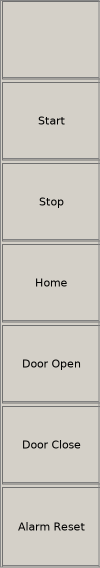
VISUALIZATION SideBar  // 100x568
    Button (2,1 99x78), colour toggle: GVL_HMI.bLpAutoMode, text list: 'TextList', text index: GVL_HMI.iTextIndex
        OnMouseClick: execute { GVL_HMI.bBtAutoMode := true; }
    Button (2,82 99x78), "Start", colour toggle: gvl_hmi.bLpStart
        OnMouseClick: execute { GVL_HMI.bBtStart := TRUE; }
    Button (2,163 99x78), "Stop", colour toggle: GVL_Status.bStopCmd
        OnMouseClick: execute { GVL_HMI.bBtStop := True; }
    Button (2,244 99x78), "Home", colour toggle: GVL_HMI.bLpHome
        OnMouseClick: execute { GVL_HMI.bBtHome := True; }
    Button (2,325 99x78), "Door Open", colour toggle: GVL_Status.bSafetyDoorUnlocked
        OnMouseClick: execute { GVL_HMI.bBtDoorUnlock := True; }
    Button (2,406 99x78), "Door Close", colour toggle: GVL_Status.bSafetyDoorLocked
        OnMouseClick: execute { GVL_HMI.bBtDoorLock := True; }
    Button (2,487 99x80), "Alarm Reset", colour toggle: gvl_hmi.bLpAlarmReset
        OnMouseClick: execute { GVL_HMI.bBtAlarmReset := True; }
END_VISUALIZATION

(* stored: Version 1.1.0.1
   Visu SideBar: Id {40bafb08-da32-41f4-a447-5b3a3fd50354} *)
